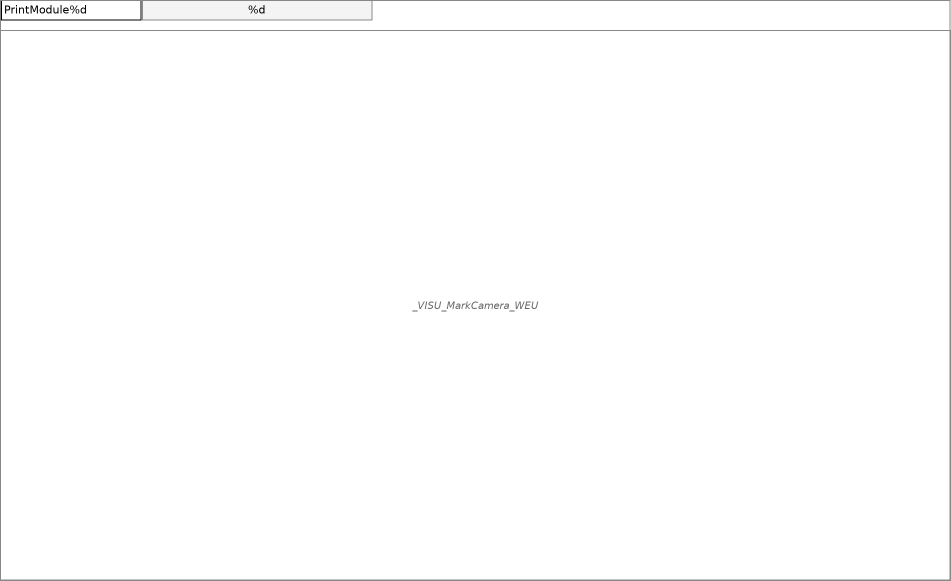
VISUALIZATION VISU_MarkCamera_WEU  // 951x581
    Frame (0,30 951x551)
        shows _VISU_MarkCamera_WEU(mCam := PRG_PRINT.fbPrintModule[PRG_PRINT.nSelectPmView].fbMarkCameraWeu, mMarkDetect := PRG_PRINT.fbPrintModule[PRG_PRINT.nSelectPmView].fbMarkDetection)
    Scrollbar (142,0 230x20), "%d", text variable: PRG_PRINT.nSelectPmView
        p1057716461: PRG_PRINT.nSelectPmView
    Rectangle (1,0 140x20), "PrintModule%d", text variable: PRG_PRINT.nSelectPmView
END_VISUALIZATION

(* stored: Version 1.1.0.1, ProductVersion 3.1.4024.11
   Visu VISU_MarkCamera_WEU: Id {35356e6c-d44b-4d0e-b2f7-2e0dcd99e062} *)
